// TIA Portal project "PPU" (V13)

(* hardware
DEVICE "S7300/ET200M-Station_1"  S7-300 station
   slot 0: "Profilschiene_0"  Rail  6ES7 390-1***0-0AA0
   slot 1: "PS 307 5A_1"  PS 307 5A  6ES7 307-1EA00-0AA0
   slot 2: "SIMATIC S7-300"  CPU 314C-2 PN/DP  6ES7 314-6EH04-0AB0  V3.3
      slot 2: "PROFINET-Schnittstelle_1"  PN-IO
         slot 1: "Port_1"  Port
         slot 2: "Port_2"  Port
      slot 5: "DI 24/DO 16_1"  DI24/DO16
      slot 6: "AI 5/AO 2_1"  AI5/AO2
      slot 7: "Zählen_1"  Counter
      slot 8: "Positionieren_1"  Positioning
   slot 4: "CP 343-2_1"  CP 343-2  6GK7 343-2AH01-0XA0  V3.1
*)

// ===== PLC "SIMATIC S7-300"  CPU 314C-2 PN/DP =====

VAR_GLOBAL   // PLC tag table "Standard-Variablentabelle"
   "Mx_StartingFlag" AT %M20.0 : Bool;   // Starting flag to activate the sequence (step 1)
   "Mb_FlagByte10" AT %MB10 : Byte;   // Flag byte 10
   "Ix_S0_OFF" AT %I124.0 : Bool;   // Stop pushbutton (NC)
   "Ix_S1_ON" AT %I124.1 : Bool;   // Start pushbutton
   "Ix_1S1_Cyl1ARet" AT %I124.2 : Bool;   // Cylinder 1A retracted
   "Ix_1S2_Cyl1AExt" AT %I124.3 : Bool;   // Cylinder 1A extended
   "Ix_2S1_Cyl2ARet" AT %I124.4 : Bool;   // Cylinder 2A retracted
   "Ix_2S2_Cyl2AExt" AT %I124.5 : Bool;   // Cylinder 2A extended
   "Qx_1M1_MoveCyl1AOut" AT %Q124.0 : Bool;   // Move package to the roller conveyer
   "Qx_1M2_MoveCyl1AIn" AT %Q124.1 : Bool;   // Move cylinder 1A in
   "Qx_2M1_MoveCyl2AOut" AT %Q124.2 : Bool;   // Move package to the roller slide
   "Qx_2M2_MoveCyl2AIn" AT %Q124.3 : Bool;   // Move cylinder 2A in
   "Qx_P1_PackageInMotion" AT %Q124.4 : Bool;   // Package in motion
   "Mx_Step0" AT %M10.0 : Bool;   // Flag Step 0
   "Mx_Step1" AT %M10.1 : Bool;   // Flag Step 1
   "Mx_Step2" AT %M10.2 : Bool;   // Flag Step 2
   "Mx_Step3" AT %M10.3 : Bool;   // Flag Step 3
   "Mx_Clock1Hz" AT %M100.5 : Bool;   // Flag Clock 1Hz
END_VAR

FUNCTION "FC1 Graphcet" : Void   // FC1, FBD
{ S7_Optimized_Access := 'FALSE' }
VERSION : 0.1
BEGIN

REGION Network 1: Step 0
   // Step 0 ist set if  the starting flag M20.0 is activated or if Both cyinders are retracted (1S1 and 1S2) and step 3 is activated. Step 0 ist resetted by step 1
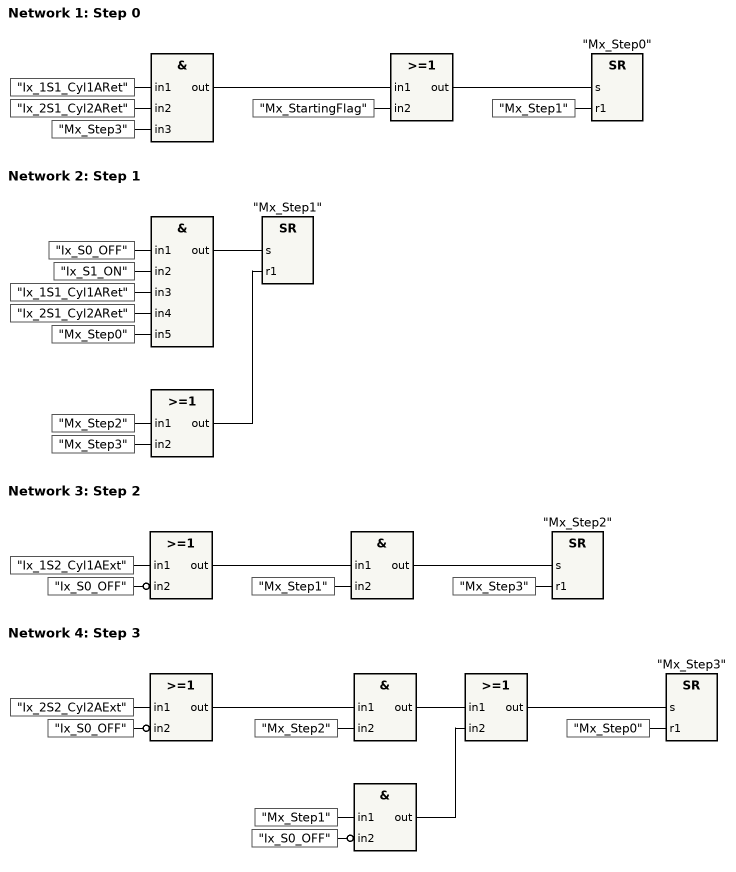
   IF ("Ix_1S1_Cyl1ARet" AND "Ix_2S1_Cyl2ARet" AND "Mx_Step3") OR "Mx_StartingFlag" THEN
       "Mx_Step0" := TRUE;   // SR flip-flop
   END_IF;
   IF "Mx_Step1" THEN "Mx_Step0" := FALSE; END_IF;
END_REGION

REGION Network 2: Step 1
   // Step 1 is set if the OFF bushbutton is not activated (S0=1), the ON pushbutton is activ(S1=1), both cylinders are retracted (1S1 and 1S2 active) and step 0 is set. step 1 is resettet by step 2 or step 3.
   IF "Ix_S0_OFF" AND "Ix_S1_ON" AND "Ix_1S1_Cyl1ARet" AND "Ix_2S1_Cyl2ARet" AND "Mx_Step0" THEN
       "Mx_Step1" := TRUE;   // SR flip-flop
   END_IF;
   IF "Mx_Step2" OR "Mx_Step3" THEN "Mx_Step1" := FALSE; END_IF;
END_REGION

REGION Network 3: Step 2
   // Step 2 is set if the cylinder 1A is extended 1S2 or the OFF pushbutton is pushed (S0=0) and the step 1 is set. Step 2 is resetted by step 3.
   IF ("Ix_1S2_Cyl1AExt" OR NOT "Ix_S0_OFF") AND "Mx_Step1" THEN
       "Mx_Step2" := TRUE;   // SR flip-flop
   END_IF;
   IF "Mx_Step3" THEN "Mx_Step2" := FALSE; END_IF;
END_REGION

REGION Network 4: Step 3
   // Step 3 is set if cylinder 2A is extended 1S2 or if the OFF pushbutton is pushed (S0=0) and step 2 is active or if stpe 1 is activ and the OFF pushbutton is pushed (S0=0) . Step 3 is resettet by step 0.
   IF (("Ix_2S2_Cyl2AExt" OR NOT "Ix_S0_OFF") AND "Mx_Step2") OR ("Mx_Step1" AND NOT "Ix_S0_OFF") THEN
       "Mx_Step3" := TRUE;   // SR flip-flop
   END_IF;
   IF "Mx_Step0" THEN "Mx_Step3" := FALSE; END_IF;
END_REGION
END_FUNCTION

FUNCTION "FC2 Actions" : Void   // FC2, FBD
{ S7_Optimized_Access := 'FALSE' }
VERSION : 0.1
BEGIN

REGION Network 1: Moving Cylinder 1A out
   // Cylinder A1 is moving out if step 1 is active.
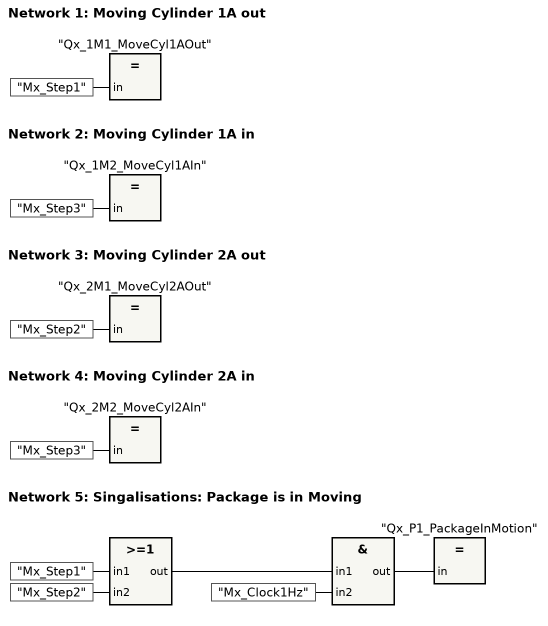
   "Qx_1M1_MoveCyl1AOut" := "Mx_Step1";
END_REGION

REGION Network 2: Moving Cylinder 1A in
   // Cylinder 1A is moving in if step 3 ist active.
   "Qx_1M2_MoveCyl1AIn" := "Mx_Step3";
END_REGION

REGION Network 3: Moving Cylinder 2A out
   // Cylinder 2A is moving out if step 2 is active.
   "Qx_2M1_MoveCyl2AOut" := "Mx_Step2";
END_REGION

REGION Network 4: Moving Cylinder 2A in
   // Cylinder 2A is moving in if step 3 is active.
   "Qx_2M2_MoveCyl2AIn" := "Mx_Step3";
END_REGION

REGION Network 5: Singalisations: Package is in Moving
   // If step 1 or step 2 is active the Lamp is flashing with 1Hz becaus of the clock M100.5
   "Qx_P1_PackageInMotion" := ("Mx_Step1" OR "Mx_Step2") AND "Mx_Clock1Hz";
END_REGION
END_FUNCTION

ORGANIZATION_BLOCK "Main"   // OB1, FBD
TITLE = "Main Program Sweep (Cycle)"
{ S7_Optimized_Access := 'FALSE' }
VERSION : 0.1
BEGIN

REGION Network 1: FC1 Graphcet
   // Calling the FC1
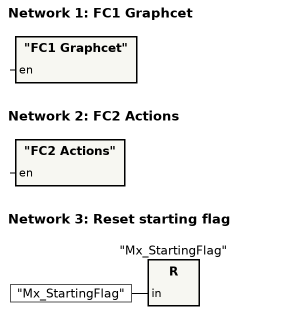
   "FC1 Graphcet"();
END_REGION

REGION Network 2: FC2 Actions
   // Calling the FC2
   "FC2 Actions"();
END_REGION

REGION Network 3: Reset starting flag
   // Resetting the starting flag
   IF "Mx_StartingFlag" THEN "Mx_StartingFlag" := FALSE; END_IF;
END_REGION
END_ORGANIZATION_BLOCK

ORGANIZATION_BLOCK "COMPLETE RESTART"   // OB100, FBD
TITLE = "Complete Restart"
{ S7_Optimized_Access := 'FALSE' }
VERSION : 0.1
BEGIN

REGION Network 1: Reset Flagbyte 10
   // Resetting all bits from the byte 10
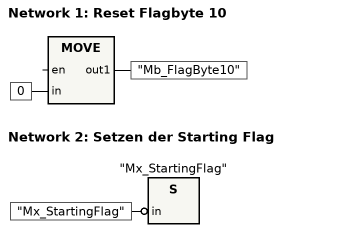
   "Mb_FlagByte10" := 0;
END_REGION

REGION Network 2: Setzen der Starting Flag
   // Setting the starting flag
   IF NOT "Mx_StartingFlag" THEN "Mx_StartingFlag" := TRUE; END_IF;
END_REGION
END_ORGANIZATION_BLOCK